(* IEC 61131-3 sources: volt/packages/volt-lsp-iec/test-corpus/awa-palletizer/Device/Plc Logic/Application/Library Manager/CmpSrv, 6 files *)

(* ---- EVTPARAM_CMPSRV.dut ---- *)
TYPE EVTPARAM_CMPSRV :
STRUCT
	PSERVICEHANDLERPARAMETER : POINTER TO SERVICEHANDLER_PARAMETER;
END_STRUCT
END_TYPE

(* ---- HEADER_TAG.dut ---- *)
TYPE HEADER_TAG :
STRUCT
	USHEADERTAG : UINT;
	USHEADERLENGTH : UINT;
	USSERVICEGROUP : UINT;
	USSERVICE : UINT;
	ULSESSIONID : UDINT;
	ULSERVICELENGTH : UDINT;
END_STRUCT
END_TYPE

(* ---- PROTOCOL_DATA_UNIT.dut ---- *)
TYPE PROTOCOL_DATA_UNIT :
STRUCT
	PDATA : POINTER TO BYTE;
	ULCOUNT : UDINT;
END_STRUCT
END_TYPE

(* ---- SERVICEHANDLER_PARAMETER.dut ---- *)
TYPE SERVICEHANDLER_PARAMETER :
STRUCT
	ULCHANNELID : UDINT;
	PHEADERTAG : POINTER TO HEADER_TAG;
	PDUDATA : PROTOCOL_DATA_UNIT;
	PDUSENDBUFFER : PROTOCOL_DATA_UNIT;
	RESULT : RTS_IEC_RESULT;
END_STRUCT
END_TYPE

(* ---- COMPONENTID.gvl ---- *)
VAR_GLOBAL
	CMPID_CMPSRV : UDINT := 16#1C;
END_VAR

(* ---- EVENTIDS.gvl ---- *)
VAR_GLOBAL
	EVTPARAMID_CMPSRV : UDINT := 16#1;
	EVTVERSION_CMPSRV : UDINT := 16#2;
END_VAR
